{attribute 'no_check'}
FUNCTION V_TO_INT : INT
VAR_INPUT
    analog : REAL;
END_VAR
VAR
    iBits :INT := 30518;
    iFullRange:INT := 10;
END_VAR

if ( iFullRange = 0 ) THEN iFullRange := 10;END_IF
V_TO_INT := REAL_TO_INT(analog * 30518 /iFullRange);

END_FUNCTION

(* stored: Version 1.1.0.1
   POU V_TO_INT: Id {13161351-f8bf-4d9a-8d5b-3b10710d601a}, SpecialFunc None *)
